// TwinCAT 3 PLC project ph_lv1_motion_savepoint
// Title: tclib_ph_lv1_motion_savepoint
// Company: Poh
// Author: Poh
// ProjectVersion: 0.1.1.0
// ProgramVersion: 3.1.4020.1
// libraries:
//   Tc2_Standard, * (Beckhoff Automation GmbH)
//   Tc2_System, * (Beckhoff Automation GmbH)
//   tclib_ph_lv0, * (Poh)
// project tree:
//   Lv1_Motion_SavePoints/ C_SAVEPOINT_RETRIVER.TcPOU, S_POSITION3D_TO_S_POSITION2D.TcPOU
//   Lv1_Motion_SavePoints/Datatypes/ S_POSITION2D.TcDUT, S_POSITION3D.TcDUT, S_SAVEPOINT.TcDUT, T_SaveSlot.TcDUT, T_SlotName.TcDUT
//   Lv1_Motion_SavePoints/Global Data/ GVL_MOTION_SAVEPOINT.TcGVL, PARAM_MOTION_SAVEPOINT.TcGVL
//   Version/ Global_Version.TcGVL
// (motion and I/O tree: see PLC project ph_lv0)
// real-time tasks:
//   TASK PlcTask: cycle T#10ms, priority 20, ADS port 350
//   TASK Fast: cycle T#3ms, priority 1, ADS port 351

// ---- Lv1_Motion_SavePoints/Datatypes/S_POSITION2D.TcDUT
TYPE S_POSITION2D :
STRUCT
	X : LREAL;
	Y : LREAL;
END_STRUCT
END_TYPE

// ---- Lv1_Motion_SavePoints/Datatypes/S_POSITION3D.TcDUT
TYPE S_POSITION3D EXTENDS S_POSITION2D :
STRUCT
	Z : LREAL;
END_STRUCT
END_TYPE

// ---- Lv1_Motion_SavePoints/Datatypes/S_SAVEPOINT.TcDUT
TYPE S_SAVEPOINT EXTENDS S_POSITION3D :
STRUCT
	NAME : T_SlotName;
END_STRUCT
END_TYPE

// ---- Lv1_Motion_SavePoints/Datatypes/T_SaveSlot.TcDUT
TYPE T_SaveSlot : UINT(1..65535); END_TYPE

// ---- Lv1_Motion_SavePoints/Datatypes/T_SlotName.TcDUT
TYPE T_SlotName : STRING(32); END_TYPE

// ---- Lv1_Motion_SavePoints/Global Data/GVL_MOTION_SAVEPOINT.TcGVL
{attribute 'qualified_only'}
VAR_GLOBAL
	_SAVED_DATA : ARRAY[1..PARAM_MOTION_SAVEPOINT.SUPPORTED_SLOTS] OF S_SAVEPOINT;
END_VAR

// ---- Lv1_Motion_SavePoints/Global Data/PARAM_MOTION_SAVEPOINT.TcGVL
{attribute 'qualified_only'}
VAR_GLOBAL CONSTANT
	SUPPORTED_SLOTS : T_SaveSlot := 300;
END_VAR

// ---- Version/Global_Version.TcGVL
{attribute 'TcGenerated'}
// This function has been automatically generated from the project information.
VAR_GLOBAL CONSTANT
	{attribute 'const_non_replaced'}
	{attribute 'linkalways'}
	stLibVersion_tclib_ph_lv1_motion_savepoint : ST_LibVersion := (iMajor := 0, iMinor := 1, iBuild := 1, iRevision := 0, sVersion := '0.1.1.0');
END_VAR

// ---- Lv1_Motion_SavePoints/C_SAVEPOINT_RETRIVER.TcPOU
FUNCTION_BLOCK C_SAVEPOINT_RETRIVER
VAR_INPUT
END_VAR
VAR_OUTPUT
END_VAR
VAR
	PTR_SAVEDATA : POINTER TO S_SAVEPOINT;
END_VAR

METHOD Recall_Position_ByName : RETURN_CODE
VAR_INPUT
	NAME : T_SlotName;
	POSITION_DATA : POINTER TO S_POSITION3D;
END_VAR
VAR 
	Slot : T_SaveSlot;
END_VAR
IF POSITION_DATA = 0 THEN
	Recall_Position_ByName := ph_lv0.LV0_RETURNCODE.RETURN_ERROR;
	RETURN;
END_IF
FOR Slot := 1 TO PARAM_MOTION_SAVEPOINT.SUPPORTED_SLOTS BY 1 DO
	IF LEN(PTR_SAVEDATA[SLOT - 1].NAME) <> LEN(NAME) THEN
		CONTINUE;
	END_IF
	IF MEMCMP(ADR(PTR_SAVEDATA[SLOT-1]),ADR(NAME), LEN(NAME)) = 0 THEN
		POSITION_DATA^ := PTR_SAVEDATA[SLOT-1];
		Recall_Position_ByName := ph_lv0.LV0_RETURNCODE.RETURN_SUCCESS;
		RETURN;
	END_IF
END_FOR
Recall_Position_ByName := 2 * ph_lv0.LV0_RETURNCODE.RETURN_ERROR;
END_METHOD

METHOD Recall_Position_BySlot : RETURN_CODE
VAR_INPUT
	SLOT : T_SaveSlot;
	POSITION_DATA : POINTER TO S_POSITION3D;
END_VAR
IF SLOT < 1 OR SLOT > THIS^.SUPPORTED_SLOT_SIZE THEN
	Recall_Position_BySlot := ph_lv0.LV0_RETURNCODE.RETURN_ERROR;
ELSE
	IF POSITION_DATA = 0 THEN
		Recall_Position_BySlot := 2 * ph_lv0.LV0_RETURNCODE.RETURN_ERROR;
	ELSE
		POSITION_DATA^ := PTR_SAVEDATA[SLOT - 1];
		Recall_Position_BySlot := ph_lv0.LV0_RETURNCODE.RETURN_SUCCESS;
	END_IF
END_IF
END_METHOD

PROPERTY SAVED_DATA : POINTER TO S_SAVEPOINT
GET
SAVED_DATA := PTR_SAVEDATA;
END_GET
SET
PTR_SAVEDATA := SAVED_DATA;
END_SET
END_PROPERTY

PROPERTY SUPPORTED_SLOT_SIZE : DINT
GET
SUPPORTED_SLOT_SIZE := PARAM_MOTION_SAVEPOINT.SUPPORTED_SLOTS;
END_GET
END_PROPERTY

END_FUNCTION_BLOCK

// ---- Lv1_Motion_SavePoints/S_POSITION3D_TO_S_POSITION2D.TcPOU
FUNCTION S_POSITION3D_TO_S_POSITION2D : S_POSITION2D
VAR_INPUT
	IN_VALUE : S_POSITION2D;
END_VAR
VAR
END_VAR

S_POSITION3D_TO_S_POSITION2D := IN_VALUE;

END_FUNCTION
